Fanuc KAREL source: NC0059.KL

-- PROVISIONAL review KL for V940-1; original PC SHA256 0ac2818ecf8166097ce4f8ced2d71e677baad737dd4fc7d91f03abeb2b119904
-- Incomplete behavior may be omitted. Consult companion uncertainty JSON. Do not deploy.
PROGRAM NC0059
%NOLOCKGROUP
-- UNRESOLVED_LOCAL_POOL 1 cells at code offset 3; source declarations unknown
-- DIRECT_LOCAL_WORD_ACCESS alone does not prove INTEGER, REAL, or BOOLEAN
BEGIN
  -- V9_CONDITION_STACK_HINT 7 bounded expression windows; static native code-base-relative target link; source arms held
  -- UNRESOLVED_PC offsets 0-8; opcodes 2B,2C,7B
  -- UNRESOLVED_PC offsets 13-20; opcodes 9D,23
  -- UNRESOLVED_PC offsets 25-42; opcodes 21,40,41,42
  -- UNRESOLVED_PC offsets 47-81; opcodes 21,2E,52,23,7A,40,41,42
  -- UNRESOLVED_PC offsets 86-110; opcodes 21,2E,52,23,7A,43
  -- UNRESOLVED_PC offsets 115-128; opcodes 21,9D,57,79
  -- UNRESOLVED_PC offsets 133-151; opcodes 21,2E,52,23
  -- UNRESOLVED_PC offsets 156-161; opcodes 7A
  -- UNRESOLVED_PC offsets 166-183; opcodes 21,40,41,42
  -- UNRESOLVED_PC offsets 188-222; opcodes 21,2E,52,23,7A,40,41,42
  -- UNRESOLVED_PC offsets 227-251; opcodes 21,2E,52,23,7A,43
  -- UNRESOLVED_PC offsets 256-269; opcodes 21,9D,57,79
  -- UNRESOLVED_PC offsets 274-292; opcodes 21,2E,52,23
  -- UNRESOLVED_PC offsets 297-302; opcodes 7A
  -- UNRESOLVED_PC offsets 307-324; opcodes 21,40,41,42
  -- UNRESOLVED_PC offsets 329-363; opcodes 21,2E,52,23,7A,40,41,42
  -- UNRESOLVED_PC offsets 368-392; opcodes 21,2E,52,23,7A,43
  -- UNRESOLVED_PC offsets 397-410; opcodes 21,9D,57,79
  -- UNRESOLVED_PC offsets 415-433; opcodes 21,2E,52,23
  -- UNRESOLVED_PC offsets 438-443; opcodes 7A
  -- UNRESOLVED_PC offsets 448-465; opcodes 21,40,41,42
  -- UNRESOLVED_PC offsets 470-504; opcodes 21,2E,52,23,7A,40,41,42
  -- UNRESOLVED_PC offsets 509-533; opcodes 21,2E,52,23,7A,43
  -- UNRESOLVED_PC offsets 538-551; opcodes 21,9D,57,79
  -- UNRESOLVED_PC offsets 556-574; opcodes 21,2E,52,23
  -- UNRESOLVED_PC offsets 579-584; opcodes 7A
  -- UNRESOLVED_PC offsets 589-606; opcodes 21,40,41,42
  -- UNRESOLVED_PC offsets 611-645; opcodes 21,2E,52,23,7A,40,41,42
  -- UNRESOLVED_PC offsets 650-674; opcodes 21,2E,52,23,7A,43
  -- UNRESOLVED_PC offsets 679-692; opcodes 21,9D,57,79
  -- UNRESOLVED_PC offsets 697-715; opcodes 21,2E,52,23
  -- UNRESOLVED_PC offsets 720-725; opcodes 7A
  -- UNRESOLVED_PC offsets 730-747; opcodes 21,40,41,42
  -- UNRESOLVED_PC offsets 752-786; opcodes 21,2E,52,23,7A,40,41,42
  -- UNRESOLVED_PC offsets 791-815; opcodes 21,2E,52,23,7A,43
  -- UNRESOLVED_PC offsets 820-833; opcodes 21,9D,57,79
  -- UNRESOLVED_PC offsets 838-856; opcodes 21,2E,52,23
  -- UNRESOLVED_PC offsets 861-866; opcodes 7A
  -- UNRESOLVED_PC offsets 871-888; opcodes 21,40,41,42
  -- UNRESOLVED_PC offsets 893-927; opcodes 21,2E,52,23,7A,40,41,42
  -- UNRESOLVED_PC offsets 932-956; opcodes 21,2E,52,23,7A,43
  -- UNRESOLVED_PC offsets 961-974; opcodes 21,9D,57,79
  -- UNRESOLVED_PC offsets 979-997; opcodes 21,2E,52,23
  -- UNRESOLVED_PC offsets 1002-1007; opcodes 7A
  -- UNRESOLVED_PC offsets 1012-1029; opcodes 21,40,41,42
  -- UNRESOLVED_PC offsets 1034-1068; opcodes 21,2E,52,23,7A,40,41,42
  -- UNRESOLVED_PC offsets 1073-1097; opcodes 21,2E,52,23,7A,43
  -- UNRESOLVED_PC offsets 1102-1116; opcodes 21,9D,52,23
  -- UNRESOLVED_PC offsets 1196-1200; opcodes 7F
  -- UNRESOLVED_PC offsets 1205-1209; opcodes 27,AA
  -- UNRESOLVED_PC offsets 1214-1218; opcodes 7F
END NC0059
